FUNCTION_BLOCK App3_StripperLevelandSeparatorLevel (* Composite Function Block Type *)
  (* Standard: 61499-2 *)
  (* Version 0.0, 2018-11-06, 4DIAC-IDE, 4DIAC-Consortium *)
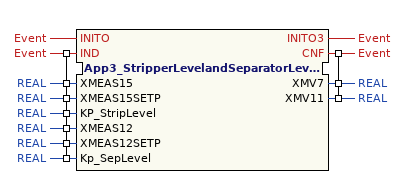
  EVENT_INPUT
    INITO; (* Initialization Request *)
    IND WITH XMEAS15, XMEAS12, XMEAS15SETP, XMEAS12SETP, KP_StripLevel, Kp_SepLevel; (* Normal Execution Request *)
  END_EVENT
  EVENT_OUTPUT
    INITO3; (* Initialization Confirm *)
    CNF WITH XMV7, XMV11; (* Execution Confirmation *)
  END_EVENT
  VAR_INPUT
    XMEAS15 : REAL;
    XMEAS15SETP : REAL;
    KP_StripLevel : REAL;
    XMEAS12 : REAL;
    XMEAS12SETP : REAL;
    Kp_SepLevel : REAL;
  END_VAR
  VAR_OUTPUT
    XMV7 : REAL;
    XMV11 : REAL;
  END_VAR
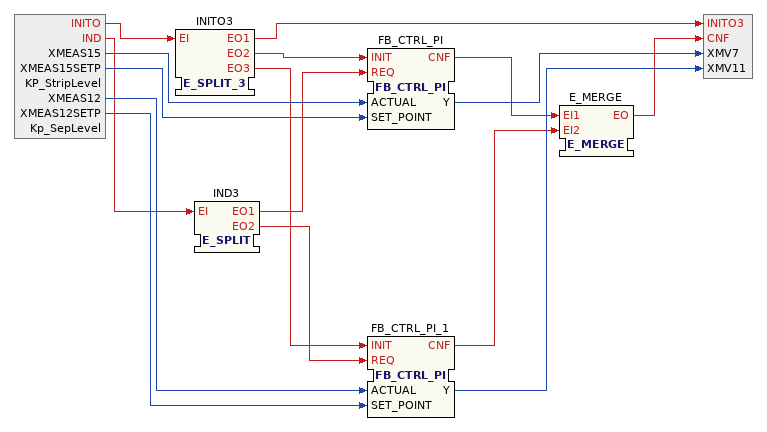
  FBS
    INITO3 : E_SPLIT_3;
    IND3 : E_SPLIT;
    E_MERGE : E_MERGE;
    FB_CTRL_PI : FB_CTRL_PI;
    FB_CTRL_PI_1 : FB_CTRL_PI;
  END_FBS
  EVENT_CONNECTIONS
    INITO TO INITO3.EI;
    INITO3.EO1 TO INITO3;
    INITO3.EO2 TO FB_CTRL_PI.INIT;
    INITO3.EO3 TO FB_CTRL_PI_1.INIT;
    IND3.EO1 TO FB_CTRL_PI.REQ;
    IND3.EO2 TO FB_CTRL_PI_1.REQ;
    FB_CTRL_PI.CNF TO E_MERGE.EI1;
    FB_CTRL_PI_1.CNF TO E_MERGE.EI2;
    E_MERGE.EO TO CNF;
    IND TO IND3.EI;
  END_CONNECTIONS
  DATA_CONNECTIONS
    FB_CTRL_PI.Y TO XMV7;
    FB_CTRL_PI_1.Y TO XMV11;
    XMEAS15 TO FB_CTRL_PI.ACTUAL;
    XMEAS15SETP TO FB_CTRL_PI.SET_POINT;
    XMEAS12 TO FB_CTRL_PI_1.ACTUAL;
    XMEAS12SETP TO FB_CTRL_PI_1.SET_POINT;
  END_CONNECTIONS
END_FUNCTION_BLOCK
